(* PLC project SFC_Evolution_4, Beckhoff Automation GmbH TwinCAT PLC Control 3.5.10.30 *)
(* stored: creationDateTime 2019-09-30T14:21:44.2564391, modificationDateTime 2019-09-30T14:21:44.2564391 *)

PROGRAM Main
VAR
	VAR_1: BOOL;
	Condition_1: BOOL;
	Condition_2: BOOL;
	Changed: BOOL;
END_VAR

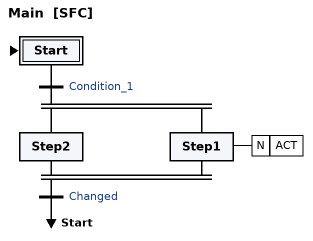
INITIAL_STEP Start:
END_STEP
TRANSITION FROM Start TO (Step2, Step1)
  := Condition_1;
END_TRANSITION
STEP Step2:
END_STEP
TRANSITION FROM (Step2, Step1) TO Start
  := Changed;
END_TRANSITION
STEP Step1:
  ACT(N);
END_STEP

ACTION ACT:
                      changed := TRUE;
                    
END_ACTION
END_PROGRAM

CONFIGURATION Application
  RESOURCE SFC_Evolution_4 ON PLC
    TASK PlcTask(INTERVAL := T#0ms, PRIORITY := 20);
    PROGRAM Main WITH PlcTask : Main;
  END_RESOURCE
END_CONFIGURATION
